ORGANIZATION_BLOCK MAIN:OB1
TITLE=Make a Logic when I0.0 is pressed, Q0.0 is ON for 10 seconds then OFF
BEGIN
Network 1
LD     I0.0
LPS
AN     T32
=      Q0.0
LPP
TON    T32, 10000
END_ORGANIZATION_BLOCK
SUBROUTINE_BLOCK SBR_0:SBR0
TITLE=SUBROUTINE COMMENTS
BEGIN
Network 1 // Network Title
// Network Comment
END_SUBROUTINE_BLOCK
INTERRUPT_BLOCK INT_0:INT0
TITLE=INTERRUPT ROUTINE COMMENTS
BEGIN
Network 1 // Network Title
// Network Comment
END_INTERRUPT_BLOCK
